PROGRAM F15_CaseControlCACData
VAR
	rtrigScanBarcode			: R_TRIG;
	fbScannerCtrl				: FB_SCANNER_CameraSelect;
	bScanCaseLabel				: BOOL;
	fbCaseLableEvaluation		: FB_SCANNER_Evaluation;

	rtrigSetCaseValidationOK	: R_TRIG;
	rtrigSetCaseValidationNOK	: R_TRIG;

	sCaseSerialCode				: T_CASE_Barcode;
	sFirstOuterInCase			: T_OUTER_Barcode;
	sLastOuterInCase			: T_OUTER_Barcode;
	sFirstPackSerialCode		: T_PACK_Barcode;
	sLastPackSerialCode			: T_PACK_Barcode;


	fbSequenceControl			: FB_SYSTEM_SeqControl;
	nSequenceStep				: INT;
	b00_Idle					: BOOL;
	b01_ScanLabel				: BOOL;
	b03_CreateFileName			: BOOL;
	b05_MoveCaseData			: BOOL;
	b08_WriteFSSFile			: BOOL;
	b10_CaseTraceValid			: BOOL;
	b18_CaseValid				: BOOL;
	b19_CaseInvalid				: BOOL;
	b20_Done					: BOOL;

	bDone						: BOOL;
	bBusy						: BOOL;
	tonScanTimeout				: TON;
	tonOverTime					: TON;

	rtrigCACData				: R_TRIG;
	tF15TimeExecution			: TIME;
	bTestSeq					: BOOL;
	sCACFileTemplate			: T_CAC_Filename;

	stValidateCACData			: ST_CAC_Data;
	fbMoveCaseData				: FB_CASE_ValidatePrintCACData;

	sPrintCaseContent			: STRING(255);

	fbPopulateCHMData				: FB_CHM_PopulateDataForFSS3;
	fbWriteCHMFile				: FB_CHM_WriteFSS3Files; (*Old system supporting FSS2 -> FB_CHM_WriteFSSFile;*)

	fbWriteCACToArchiveDB			: FB_CAC_WriteHierachyToDB;
	fbCaseStatusPulse				: TON;
	bCACValid					: BOOL;
	bCHMValid					: BOOL;


	fbMoveVerifiedCAC				: FB_CASE_MoveVerifiedCAC;
	fbMoveFailedCAC				: FB_CASE_MoveFailedCAC;

	fbCaseEfficiency				: FB_KPI_GenericEfficiency;
	fbCaseInspectionEfficiency		: FB_KPI_CaseEfficiency;
	(*fbCaseInspectionEfficiency		: FB_KPI_PACAN_CaseEfficiency;*)
	fbRejectCount					: CTU;
	nRejectActualCount				: WORD;

	fbCaseValidationScanned			: FB_CTU32;
	fbCaseValidationCorrect			: FB_CTU32;
	fbCaseValidationNoCaseLabel		: FB_CTU32;
	fbCaseValidationCasePackerReject	: FB_CTU32;

	aLastCaseBarcodes				: ARRAY[1..cMAX_LAST_CASE_BARCODES] OF T_CASE_Barcode;
	fbAddVerifiedCaseBarcode		: FB_CASE_AddVerifiedCaseBarcode;

	fbCaseLevelCounter	: FB_KPI_CaseLevelCounter;
	tofCaseValidationCameraOFFDelay 	: TOF;

	fbFileWriteCACError				: FB_LOG_FileWriteError;
	fbFileWriteCHMError			: FB_LOG_FileWriteError;

END_VAR
(*
VAR CONSTANT
	sOptions						: ST_SCANNER_Options := (eScannerType := E_MV_440SR_FULL, nImageBuffer := 1, nExpectedResp := 1);
END_VAR*)
VAR // added by the converter: edge detectors and wires of the graphical bodies
    _w1, _w2, _w3, _w4 : BOOL;
END_VAR

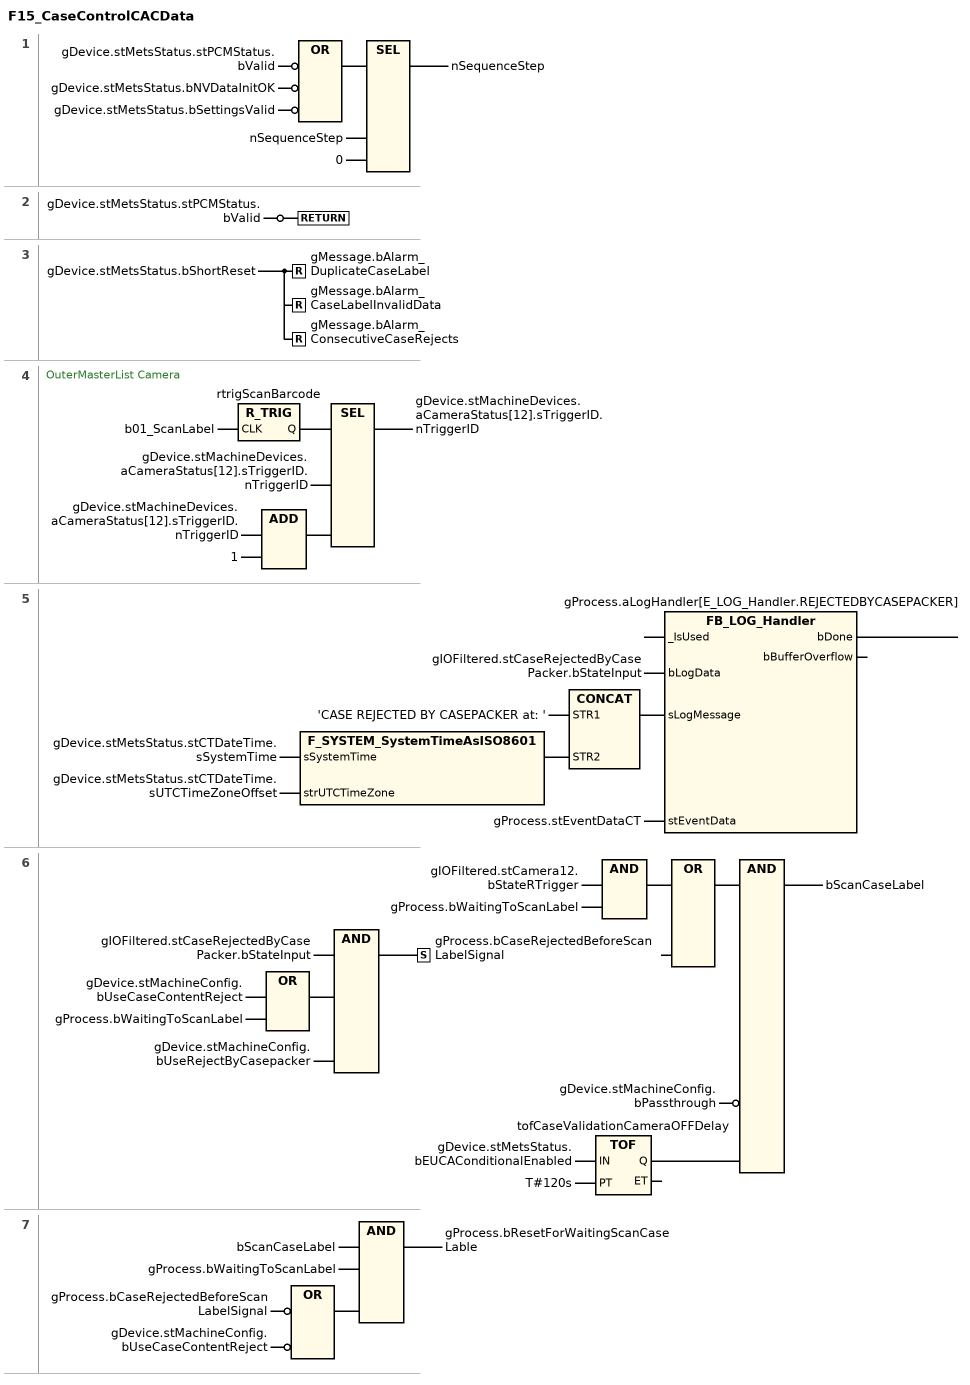
// NETWORK 1
nSequenceStep := SEL(NOT gDevice.stMetsStatus.stPCMStatus.bValid OR NOT gDevice.stMetsStatus.bNVDataInitOK OR NOT gDevice.stMetsStatus.bSettingsValid, nSequenceStep, 0);

// NETWORK 2
IF NOT gDevice.stMetsStatus.stPCMStatus.bValid THEN RETURN; END_IF

// NETWORK 3
gMessage.bAlarm_DuplicateCaseLabel R= gDevice.stMetsStatus.bShortReset;
gMessage.bAlarm_CaseLabelInvalidData R= gDevice.stMetsStatus.bShortReset;
gMessage.bAlarm_ConsecutiveCaseRejects R= gDevice.stMetsStatus.bShortReset;

// NETWORK 4
// OuterMasterList Camera
rtrigScanBarcode(CLK := b01_ScanLabel); // R_TRIG
gDevice.stMachineDevices.aCameraStatus[12].sTriggerID.nTriggerID := SEL(rtrigScanBarcode.Q, gDevice.stMachineDevices.aCameraStatus[12].sTriggerID.nTriggerID, gDevice.stMachineDevices.aCameraStatus[12].sTriggerID.nTriggerID + 1);

// NETWORK 5
gProcess.aLogHandler[E_LOG_Handler.REJECTEDBYCASEPACKER](
    bLogData := gIOFiltered.stCaseRejectedByCasePacker.bStateInput,
    sLogMessage := CONCAT(STR1 := 'CASE REJECTED BY CASEPACKER at: ', STR2 := F_SYSTEM_SystemTimeAsISO8601(sSystemTime := gDevice.stMetsStatus.stCTDateTime.sSystemTime, strUTCTimeZone := gDevice.stMetsStatus.stCTDateTime.sUTCTimeZoneOffset)),
    stEventData := gProcess.stEventDataCT); // FB_LOG_Handler

// NETWORK 6
_w2 := gIOFiltered.stCamera12.bStateRTrigger AND gProcess.bWaitingToScanLabel;
_w1 := gIOFiltered.stCaseRejectedByCasePacker.bStateInput AND (gDevice.stMachineConfig.bUseCaseContentReject OR gProcess.bWaitingToScanLabel) AND gDevice.stMachineConfig.bUseRejectByCasepacker;
gProcess.bCaseRejectedBeforeScanLabelSignal S= _w1;
tofCaseValidationCameraOFFDelay(IN := gDevice.stMetsStatus.bEUCAConditionalEnabled, PT := T#120s); // TOF
bScanCaseLabel := (_w2 OR _w1) AND NOT gDevice.stMachineConfig.bPassthrough AND tofCaseValidationCameraOFFDelay.Q;

// NETWORK 7
gProcess.bResetForWaitingScanCaseLable := bScanCaseLabel AND gProcess.bWaitingToScanLabel AND (NOT gProcess.bCaseRejectedBeforeScanLabelSignal OR NOT gDevice.stMachineConfig.bUseCaseContentReject);

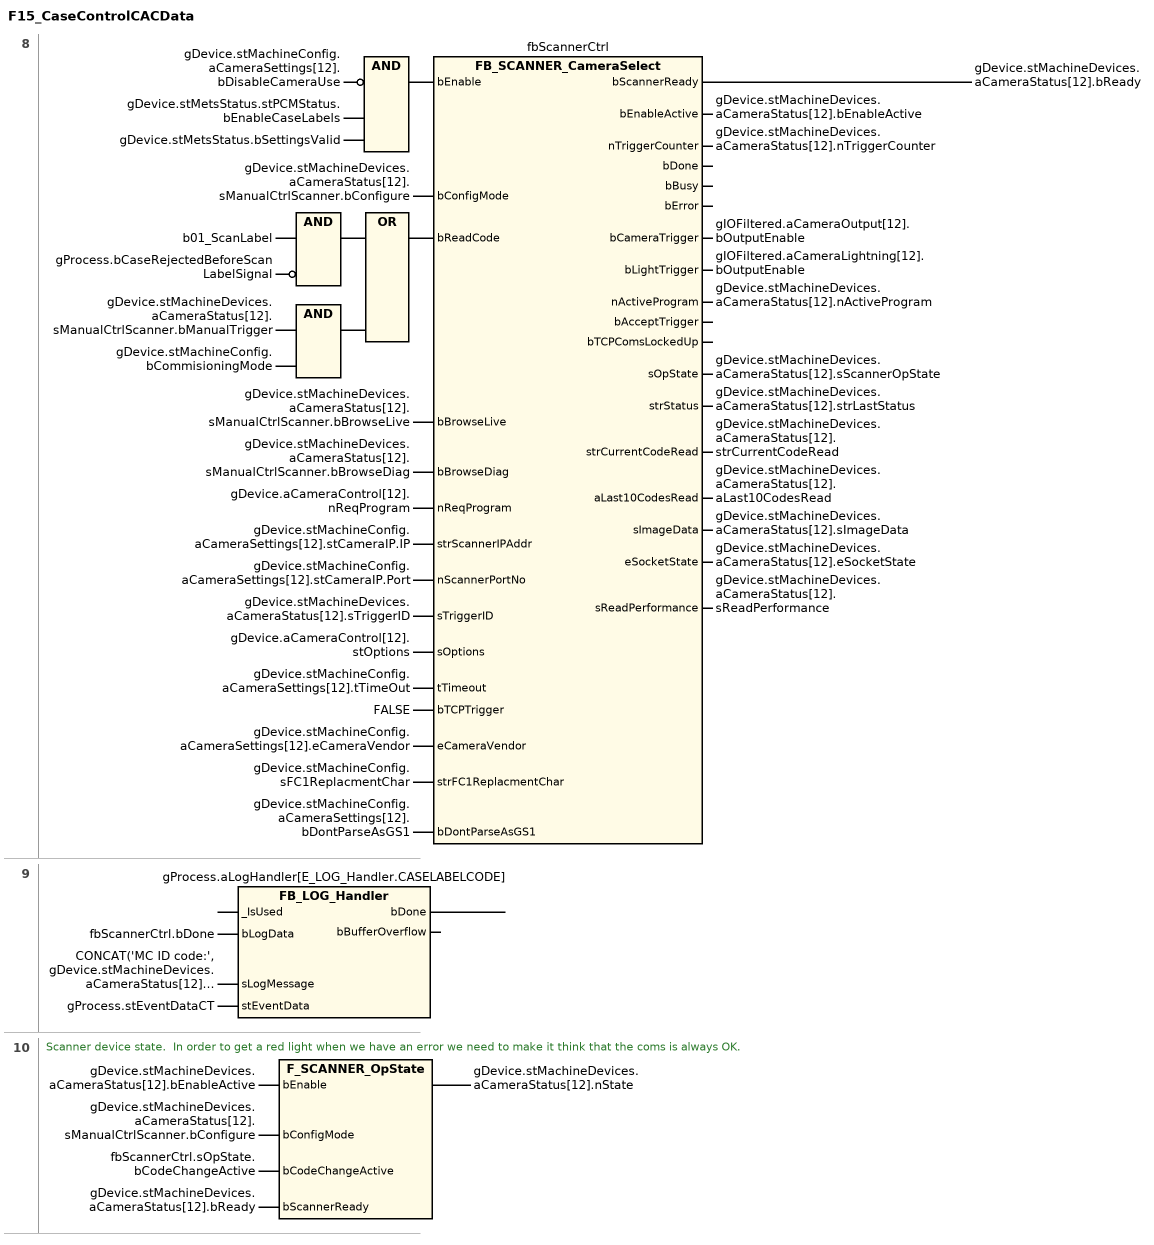
// NETWORK 8
fbScannerCtrl(
    bEnable := NOT gDevice.stMachineConfig.aCameraSettings[12].bDisableCameraUse AND gDevice.stMetsStatus.stPCMStatus.bEnableCaseLabels AND gDevice.stMetsStatus.bSettingsValid,
    bConfigMode := gDevice.stMachineDevices.aCameraStatus[12].sManualCtrlScanner.bConfigure,
    bReadCode := b01_ScanLabel AND NOT gProcess.bCaseRejectedBeforeScanLabelSignal OR gDevice.stMachineDevices.aCameraStatus[12].sManualCtrlScanner.bManualTrigger AND gDevice.stMachineConfig.bCommisioningMode,
    bBrowseLive := gDevice.stMachineDevices.aCameraStatus[12].sManualCtrlScanner.bBrowseLive,
    bBrowseDiag := gDevice.stMachineDevices.aCameraStatus[12].sManualCtrlScanner.bBrowseDiag,
    nReqProgram := gDevice.aCameraControl[12].nReqProgram,
    strScannerIPAddr := gDevice.stMachineConfig.aCameraSettings[12].stCameraIP.IP,
    nScannerPortNo := gDevice.stMachineConfig.aCameraSettings[12].stCameraIP.Port,
    sTriggerID := gDevice.stMachineDevices.aCameraStatus[12].sTriggerID,
    sOptions := gDevice.aCameraControl[12].stOptions,
    tTimeout := gDevice.stMachineConfig.aCameraSettings[12].tTimeOut,
    bTCPTrigger := FALSE,
    eCameraVendor := gDevice.stMachineConfig.aCameraSettings[12].eCameraVendor,
    strFC1ReplacmentChar := gDevice.stMachineConfig.sFC1ReplacmentChar,
    bDontParseAsGS1 := gDevice.stMachineConfig.aCameraSettings[12].bDontParseAsGS1,
    bEnableActive => gDevice.stMachineDevices.aCameraStatus[12].bEnableActive,
    nTriggerCounter => gDevice.stMachineDevices.aCameraStatus[12].nTriggerCounter,
    bCameraTrigger => gIOFiltered.aCameraOutput[12].bOutputEnable,
    bLightTrigger => gIOFiltered.aCameraLightning[12].bOutputEnable,
    nActiveProgram => gDevice.stMachineDevices.aCameraStatus[12].nActiveProgram,
    sOpState => gDevice.stMachineDevices.aCameraStatus[12].sScannerOpState,
    strStatus => gDevice.stMachineDevices.aCameraStatus[12].strLastStatus,
    strCurrentCodeRead => gDevice.stMachineDevices.aCameraStatus[12].strCurrentCodeRead,
    aLast10CodesRead => gDevice.stMachineDevices.aCameraStatus[12].aLast10CodesRead,
    sImageData => gDevice.stMachineDevices.aCameraStatus[12].sImageData,
    eSocketState => gDevice.stMachineDevices.aCameraStatus[12].eSocketState,
    sReadPerformance => gDevice.stMachineDevices.aCameraStatus[12].sReadPerformance); // FB_SCANNER_CameraSelect
gDevice.stMachineDevices.aCameraStatus[12].bReady := fbScannerCtrl.bScannerReady;

// NETWORK 9
gProcess.aLogHandler[E_LOG_Handler.CASELABELCODE](
    bLogData := fbScannerCtrl.bDone,
    sLogMessage := CONCAT('MC ID code:', gDevice.stMachineDevices.aCameraStatus[12].strCurrentCodeRead),
    stEventData := gProcess.stEventDataCT); // FB_LOG_Handler

// NETWORK 10
// Scanner device state.  In order to get a red light when we have an error we need to make it think that the coms is always OK.
gDevice.stMachineDevices.aCameraStatus[12].nState := F_SCANNER_OpState(bEnable := gDevice.stMachineDevices.aCameraStatus[12].bEnableActive, bConfigMode := gDevice.stMachineDevices.aCameraStatus[12].sManualCtrlScanner.bConfigure, bCodeChangeActive := fbScannerCtrl.sOpState.bCodeChangeActive, bScannerReady := gDevice.stMachineDevices.aCameraStatus[12].bReady);

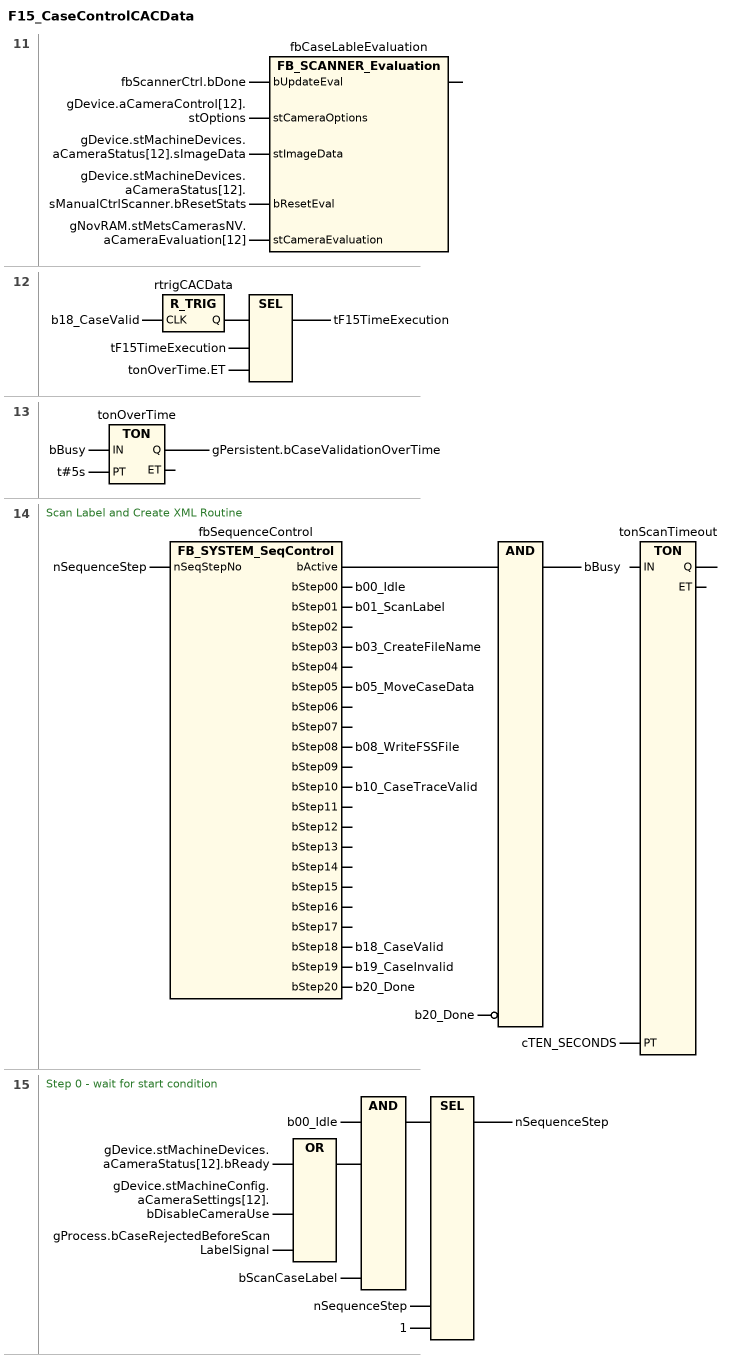
// NETWORK 11
fbCaseLableEvaluation(
    bUpdateEval := fbScannerCtrl.bDone,
    stCameraOptions := gDevice.aCameraControl[12].stOptions,
    stImageData := gDevice.stMachineDevices.aCameraStatus[12].sImageData,
    bResetEval := gDevice.stMachineDevices.aCameraStatus[12].sManualCtrlScanner.bResetStats,
    stCameraEvaluation := gNovRAM.stMetsCamerasNV.aCameraEvaluation[12]); // FB_SCANNER_Evaluation

// NETWORK 12
rtrigCACData(CLK := b18_CaseValid); // R_TRIG
tF15TimeExecution := SEL(rtrigCACData.Q, tF15TimeExecution, tonOverTime.ET);

// NETWORK 13
tonOverTime(IN := bBusy, PT := t#5s); // TON
gPersistent.bCaseValidationOverTime := tonOverTime.Q;

// NETWORK 14
// 					Scan Label and Create XML Routine
//
//
//
fbSequenceControl(
    nSeqStepNo := nSequenceStep,
    bStep00 => b00_Idle,
    bStep01 => b01_ScanLabel,
    bStep03 => b03_CreateFileName,
    bStep05 => b05_MoveCaseData,
    bStep08 => b08_WriteFSSFile,
    bStep10 => b10_CaseTraceValid,
    bStep18 => b18_CaseValid,
    bStep19 => b19_CaseInvalid,
    bStep20 => b20_Done); // FB_SYSTEM_SeqControl
_w3 := fbSequenceControl.bActive AND NOT b20_Done;
bBusy := _w3;
tonScanTimeout(IN := _w3, PT := cTEN_SECONDS); // TON

// NETWORK 15
// 					Step 0 - wait for start condition
//
//
nSequenceStep := SEL(b00_Idle AND (gDevice.stMachineDevices.aCameraStatus[12].bReady OR gDevice.stMachineConfig.aCameraSettings[12].bDisableCameraUse OR gProcess.bCaseRejectedBeforeScanLabelSignal) AND bScanCaseLabel, nSequenceStep, 1);

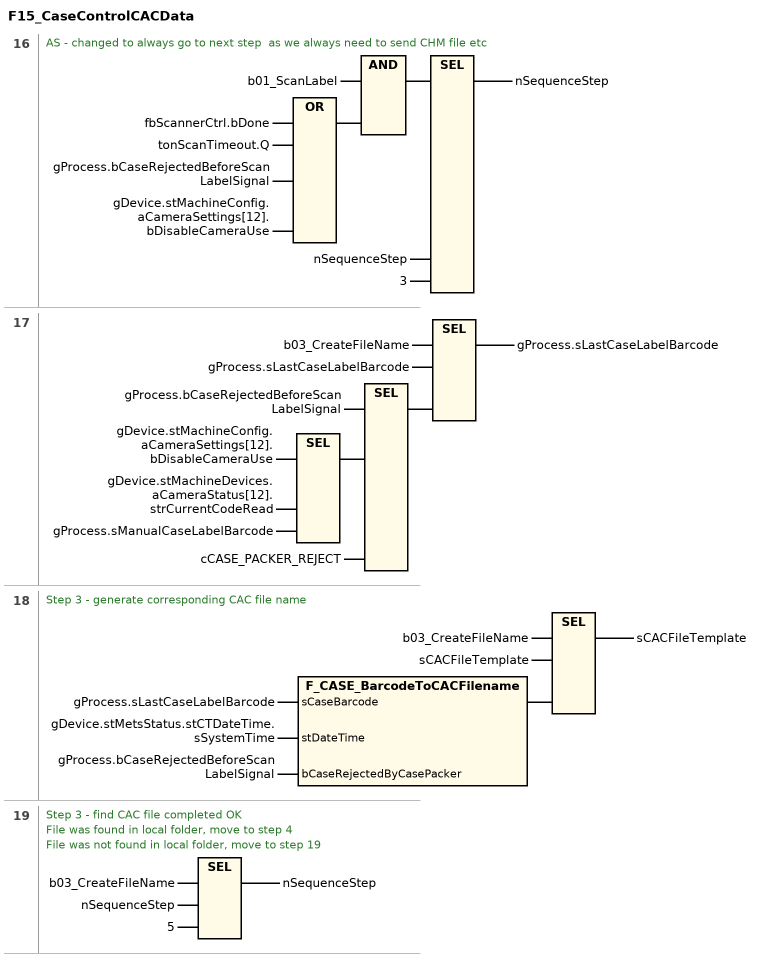
// NETWORK 16
// 					AS - changed to always go to next step  as we always need to send CHM file etc
//
//
nSequenceStep := SEL(b01_ScanLabel AND (fbScannerCtrl.bDone OR tonScanTimeout.Q OR gProcess.bCaseRejectedBeforeScanLabelSignal OR gDevice.stMachineConfig.aCameraSettings[12].bDisableCameraUse), nSequenceStep, 3);

// NETWORK 17
gProcess.sLastCaseLabelBarcode := SEL(b03_CreateFileName, gProcess.sLastCaseLabelBarcode, SEL(gProcess.bCaseRejectedBeforeScanLabelSignal, SEL(gDevice.stMachineConfig.aCameraSettings[12].bDisableCameraUse, gDevice.stMachineDevices.aCameraStatus[12].strCurrentCodeRead, gProcess.sManualCaseLabelBarcode), cCASE_PACKER_REJECT));

// NETWORK 18
// Step 3 - generate corresponding CAC file name
sCACFileTemplate := SEL(b03_CreateFileName, sCACFileTemplate, F_CASE_BarcodeToCACFilename(sCaseBarcode := gProcess.sLastCaseLabelBarcode, stDateTime := gDevice.stMetsStatus.stCTDateTime.sSystemTime, bCaseRejectedByCasePacker := gProcess.bCaseRejectedBeforeScanLabelSignal));

// NETWORK 19
// 					Step 3 - find CAC file completed OK
// File was found in local folder, move to step 4
// File was not found in local folder, move to step 19
//
nSequenceStep := SEL(b03_CreateFileName, nSequenceStep, 5);

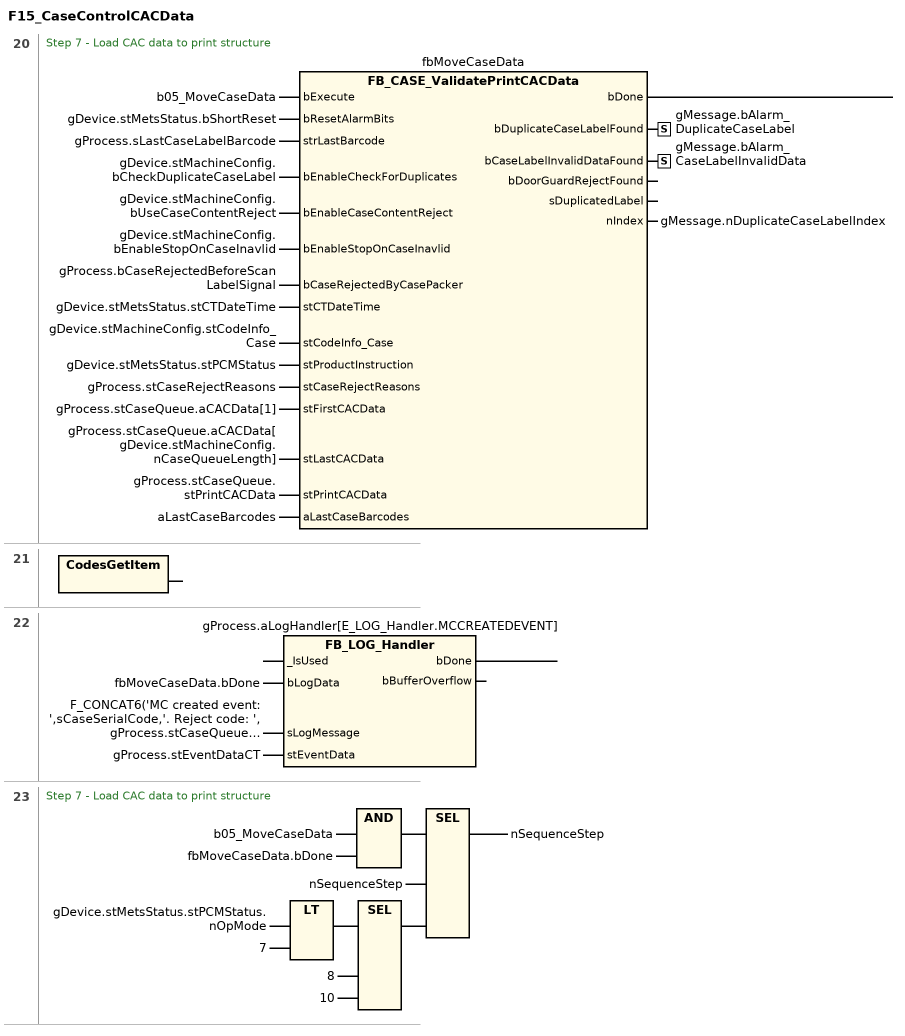
// NETWORK 20
// Step 7 - Load CAC data to print structure
fbMoveCaseData(
    bExecute := b05_MoveCaseData,
    bResetAlarmBits := gDevice.stMetsStatus.bShortReset,
    strLastBarcode := gProcess.sLastCaseLabelBarcode,
    bEnableCheckForDuplicates := gDevice.stMachineConfig.bCheckDuplicateCaseLabel,
    bEnableCaseContentReject := gDevice.stMachineConfig.bUseCaseContentReject,
    bEnableStopOnCaseInavlid := gDevice.stMachineConfig.bEnableStopOnCaseInavlid,
    bCaseRejectedByCasePacker := gProcess.bCaseRejectedBeforeScanLabelSignal,
    stCTDateTime := gDevice.stMetsStatus.stCTDateTime,
    stCodeInfo_Case := gDevice.stMachineConfig.stCodeInfo_Case,
    stProductInstruction := gDevice.stMetsStatus.stPCMStatus,
    stCaseRejectReasons := gProcess.stCaseRejectReasons,
    stFirstCACData := gProcess.stCaseQueue.aCACData[1],
    stLastCACData := gProcess.stCaseQueue.aCACData[gDevice.stMachineConfig.nCaseQueueLength],
    stPrintCACData := gProcess.stCaseQueue.stPrintCACData,
    aLastCaseBarcodes := aLastCaseBarcodes,
    nIndex => gMessage.nDuplicateCaseLabelIndex); // FB_CASE_ValidatePrintCACData
gMessage.bAlarm_DuplicateCaseLabel S= fbMoveCaseData.bDuplicateCaseLabelFound;
gMessage.bAlarm_CaseLabelInvalidData S= fbMoveCaseData.bCaseLabelInvalidDataFound;

// NETWORK 21
CodesGetItem();

// NETWORK 22
gProcess.aLogHandler[E_LOG_Handler.MCCREATEDEVENT](
    bLogData := fbMoveCaseData.bDone,
    sLogMessage := F_CONCAT6('MC created event: ',sCaseSerialCode,'. Reject code: ', gProcess.stCaseQueue.stPrintCACData.CaseRejectCode,', with case content: ', sPrintCaseContent),
    stEventData := gProcess.stEventDataCT); // FB_LOG_Handler

// NETWORK 23
// 					Step 7 - Load CAC data to print structure
//
//
nSequenceStep := SEL(b05_MoveCaseData AND fbMoveCaseData.bDone, nSequenceStep, SEL(gDevice.stMetsStatus.stPCMStatus.nOpMode < 7, 8, 10));

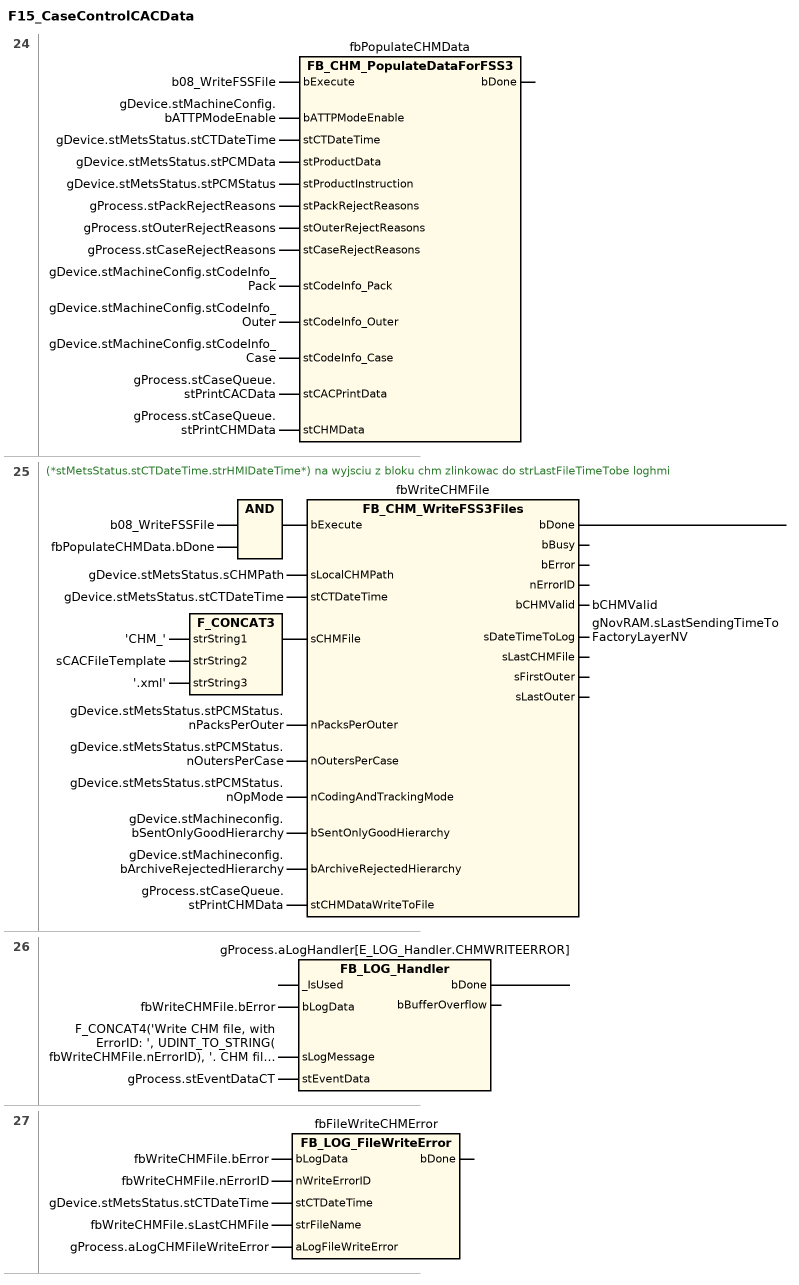
// NETWORK 24
fbPopulateCHMData(
    bExecute := b08_WriteFSSFile,
    bATTPModeEnable := gDevice.stMachineConfig.bATTPModeEnable,
    stCTDateTime := gDevice.stMetsStatus.stCTDateTime,
    stProductData := gDevice.stMetsStatus.stPCMData,
    stProductInstruction := gDevice.stMetsStatus.stPCMStatus,
    stPackRejectReasons := gProcess.stPackRejectReasons,
    stOuterRejectReasons := gProcess.stOuterRejectReasons,
    stCaseRejectReasons := gProcess.stCaseRejectReasons,
    stCodeInfo_Pack := gDevice.stMachineConfig.stCodeInfo_Pack,
    stCodeInfo_Outer := gDevice.stMachineConfig.stCodeInfo_Outer,
    stCodeInfo_Case := gDevice.stMachineConfig.stCodeInfo_Case,
    stCACPrintData := gProcess.stCaseQueue.stPrintCACData,
    stCHMData := gProcess.stCaseQueue.stPrintCHMData); // FB_CHM_PopulateDataForFSS3

// NETWORK 25
// (*stMetsStatus.stCTDateTime.strHMIDateTime*) na wyjsciu z bloku chm zlinkowac do strLastFileTimeTobe loghmi
fbWriteCHMFile(
    bExecute := b08_WriteFSSFile AND fbPopulateCHMData.bDone,
    sLocalCHMPath := gDevice.stMetsStatus.sCHMPath,
    stCTDateTime := gDevice.stMetsStatus.stCTDateTime,
    sCHMFile := F_CONCAT3(strString1 := 'CHM_', strString2 := sCACFileTemplate, strString3 := '.xml'),
    nPacksPerOuter := gDevice.stMetsStatus.stPCMStatus.nPacksPerOuter,
    nOutersPerCase := gDevice.stMetsStatus.stPCMStatus.nOutersPerCase,
    nCodingAndTrackingMode := gDevice.stMetsStatus.stPCMStatus.nOpMode,
    bSentOnlyGoodHierarchy := gDevice.stMachineconfig.bSentOnlyGoodHierarchy,
    bArchiveRejectedHierarchy := gDevice.stMachineconfig.bArchiveRejectedHierarchy,
    stCHMDataWriteToFile := gProcess.stCaseQueue.stPrintCHMData,
    bCHMValid => bCHMValid,
    sDateTimeToLog => gNovRAM.sLastSendingTimeToFactoryLayerNV); // FB_CHM_WriteFSS3Files

// NETWORK 26
gProcess.aLogHandler[E_LOG_Handler.CHMWRITEERROR](
    bLogData := fbWriteCHMFile.bError,
    sLogMessage := F_CONCAT4('Write CHM file, with ErrorID: ', UDINT_TO_STRING(fbWriteCHMFile.nErrorID), '. CHM file name: ', fbWriteCHMFile.sCHMFile),
    stEventData := gProcess.stEventDataCT); // FB_LOG_Handler

// NETWORK 27
fbFileWriteCHMError(
    bLogData := fbWriteCHMFile.bError,
    nWriteErrorID := fbWriteCHMFile.nErrorID,
    stCTDateTime := gDevice.stMetsStatus.stCTDateTime,
    strFileName := fbWriteCHMFile.sLastCHMFile,
    aLogFileWriteError := gProcess.aLogCHMFileWriteError); // FB_LOG_FileWriteError

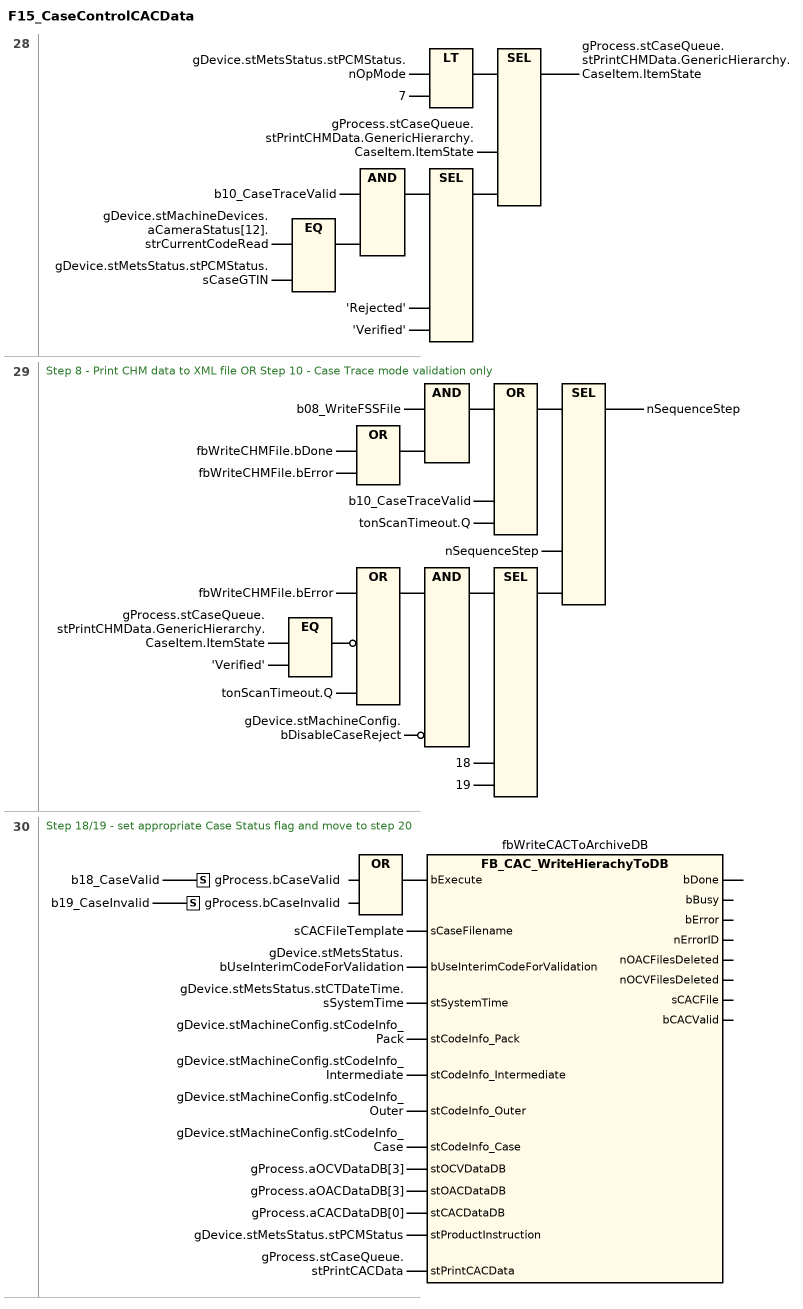
// NETWORK 28
gProcess.stCaseQueue.stPrintCHMData.GenericHierarchy.CaseItem.ItemState := SEL(gDevice.stMetsStatus.stPCMStatus.nOpMode < 7, gProcess.stCaseQueue.stPrintCHMData.GenericHierarchy.CaseItem.ItemState, SEL(b10_CaseTraceValid AND gDevice.stMachineDevices.aCameraStatus[12].strCurrentCodeRead = gDevice.stMetsStatus.stPCMStatus.sCaseGTIN, 'Rejected', 'Verified'));

// NETWORK 29
// Step 8 - Print CHM data to XML file OR Step 10 - Case Trace mode validation only
nSequenceStep := SEL(b08_WriteFSSFile AND (fbWriteCHMFile.bDone OR fbWriteCHMFile.bError) OR b10_CaseTraceValid OR tonScanTimeout.Q, nSequenceStep, SEL((fbWriteCHMFile.bError OR NOT (gProcess.stCaseQueue.stPrintCHMData.GenericHierarchy.CaseItem.ItemState = 'Verified') OR tonScanTimeout.Q) AND NOT gDevice.stMachineConfig.bDisableCaseReject, 18, 19));

// NETWORK 30
// Step 18/19 - set appropriate Case Status flag and move to step 20
gProcess.bCaseValid S= b18_CaseValid;
gProcess.bCaseInvalid S= b19_CaseInvalid;
fbWriteCACToArchiveDB(
    bExecute := b18_CaseValid OR b19_CaseInvalid,
    sCaseFilename := sCACFileTemplate,
    bUseInterimCodeForValidation := gDevice.stMetsStatus.bUseInterimCodeForValidation,
    stSystemTime := gDevice.stMetsStatus.stCTDateTime.sSystemTime,
    stCodeInfo_Pack := gDevice.stMachineConfig.stCodeInfo_Pack,
    stCodeInfo_Intermediate := gDevice.stMachineConfig.stCodeInfo_Intermediate,
    stCodeInfo_Outer := gDevice.stMachineConfig.stCodeInfo_Outer,
    stCodeInfo_Case := gDevice.stMachineConfig.stCodeInfo_Case,
    stOCVDataDB := gProcess.aOCVDataDB[3],
    stOACDataDB := gProcess.aOACDataDB[3],
    stCACDataDB := gProcess.aCACDataDB[0],
    stProductInstruction := gDevice.stMetsStatus.stPCMStatus,
    stPrintCACData := gProcess.stCaseQueue.stPrintCACData); // FB_CAC_WriteHierachyToDB

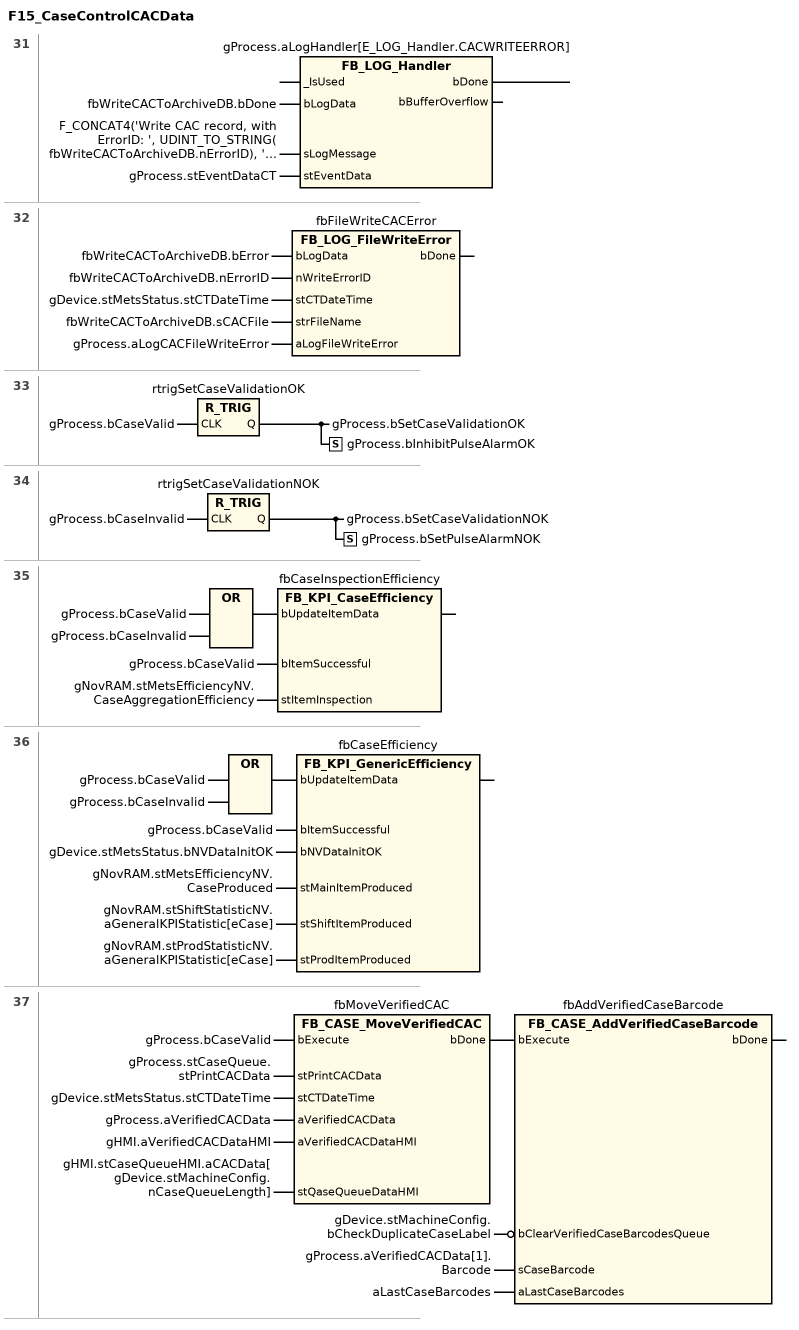
// NETWORK 31
gProcess.aLogHandler[E_LOG_Handler.CACWRITEERROR](
    bLogData := fbWriteCACToArchiveDB.bDone,
    sLogMessage := F_CONCAT4('Write CAC record, with ErrorID: ', UDINT_TO_STRING(fbWriteCACToArchiveDB.nErrorID), '. CAC file name: ', fbWriteCACToArchiveDB.sCACFile),
    stEventData := gProcess.stEventDataCT); // FB_LOG_Handler

// NETWORK 32
fbFileWriteCACError(
    bLogData := fbWriteCACToArchiveDB.bError,
    nWriteErrorID := fbWriteCACToArchiveDB.nErrorID,
    stCTDateTime := gDevice.stMetsStatus.stCTDateTime,
    strFileName := fbWriteCACToArchiveDB.sCACFile,
    aLogFileWriteError := gProcess.aLogCACFileWriteError); // FB_LOG_FileWriteError

// NETWORK 33
rtrigSetCaseValidationOK(CLK := gProcess.bCaseValid); // R_TRIG
gProcess.bSetCaseValidationOK := rtrigSetCaseValidationOK.Q;
gProcess.bInhibitPulseAlarmOK S= rtrigSetCaseValidationOK.Q;

// NETWORK 34
rtrigSetCaseValidationNOK(CLK := gProcess.bCaseInvalid); // R_TRIG
gProcess.bSetCaseValidationNOK := rtrigSetCaseValidationNOK.Q;
gProcess.bSetPulseAlarmNOK S= rtrigSetCaseValidationNOK.Q;

// NETWORK 35
fbCaseInspectionEfficiency(
    bUpdateItemData := gProcess.bCaseValid OR gProcess.bCaseInvalid,
    bItemSuccessful := gProcess.bCaseValid,
    stItemInspection := gNovRAM.stMetsEfficiencyNV.CaseAggregationEfficiency); // FB_KPI_CaseEfficiency

// NETWORK 36
fbCaseEfficiency(
    bUpdateItemData := gProcess.bCaseValid OR gProcess.bCaseInvalid,
    bItemSuccessful := gProcess.bCaseValid,
    bNVDataInitOK := gDevice.stMetsStatus.bNVDataInitOK,
    stMainItemProduced := gNovRAM.stMetsEfficiencyNV.CaseProduced,
    stShiftItemProduced := gNovRAM.stShiftStatisticNV.aGeneralKPIStatistic[eCase],
    stProdItemProduced := gNovRAM.stProdStatisticNV.aGeneralKPIStatistic[eCase]); // FB_KPI_GenericEfficiency

// NETWORK 37
fbMoveVerifiedCAC(
    bExecute := gProcess.bCaseValid,
    stPrintCACData := gProcess.stCaseQueue.stPrintCACData,
    stCTDateTime := gDevice.stMetsStatus.stCTDateTime,
    aVerifiedCACData := gProcess.aVerifiedCACData,
    aVerifiedCACDataHMI := gHMI.aVerifiedCACDataHMI,
    stQaseQueueDataHMI := gHMI.stCaseQueueHMI.aCACData[gDevice.stMachineConfig.nCaseQueueLength]); // FB_CASE_MoveVerifiedCAC
fbAddVerifiedCaseBarcode(
    bExecute := fbMoveVerifiedCAC.bDone,
    bClearVerifiedCaseBarcodesQueue := NOT gDevice.stMachineConfig.bCheckDuplicateCaseLabel,
    sCaseBarcode := gProcess.aVerifiedCACData[1].Barcode,
    aLastCaseBarcodes := aLastCaseBarcodes); // FB_CASE_AddVerifiedCaseBarcode

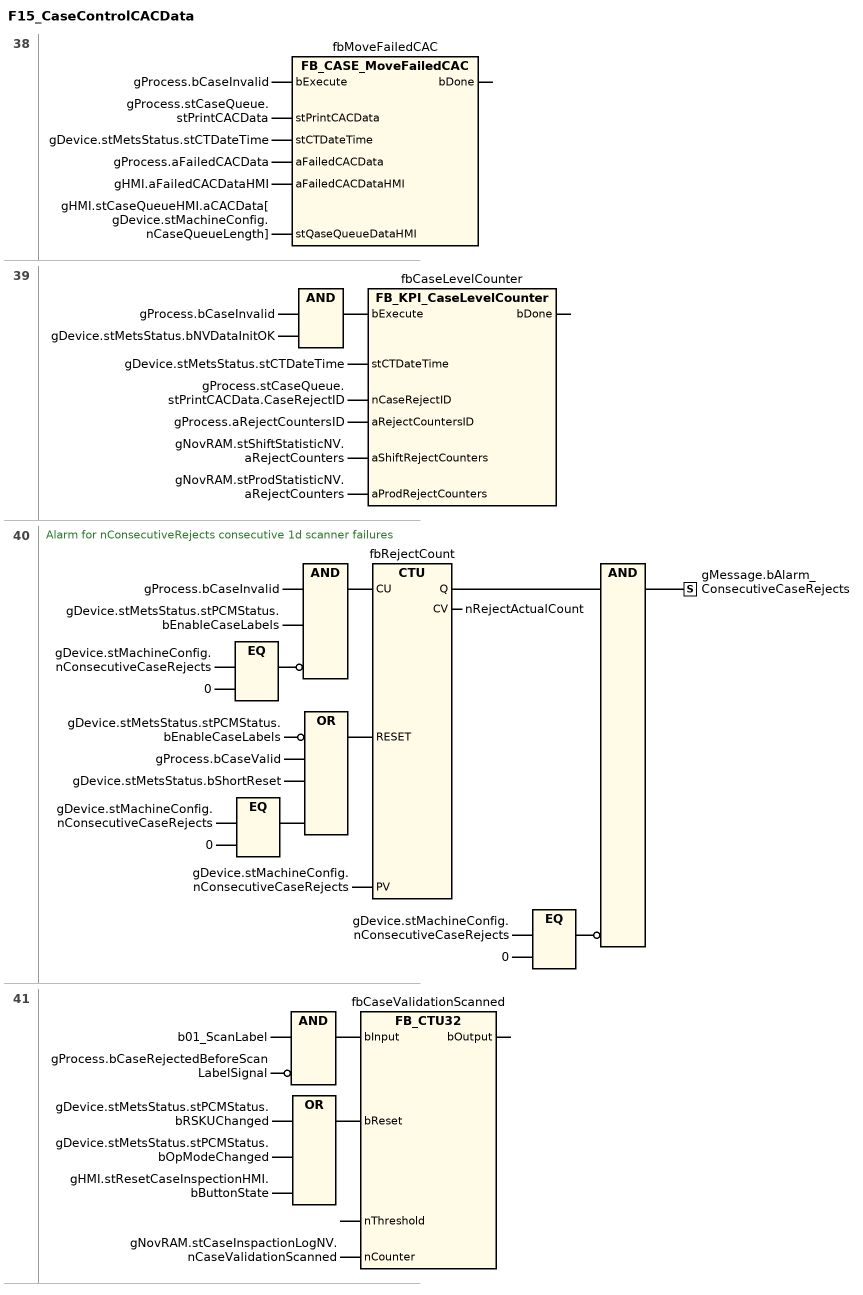
// NETWORK 38
fbMoveFailedCAC(
    bExecute := gProcess.bCaseInvalid,
    stPrintCACData := gProcess.stCaseQueue.stPrintCACData,
    stCTDateTime := gDevice.stMetsStatus.stCTDateTime,
    aFailedCACData := gProcess.aFailedCACData,
    aFailedCACDataHMI := gHMI.aFailedCACDataHMI,
    stQaseQueueDataHMI := gHMI.stCaseQueueHMI.aCACData[gDevice.stMachineConfig.nCaseQueueLength]); // FB_CASE_MoveFailedCAC

// NETWORK 39
fbCaseLevelCounter(
    bExecute := gProcess.bCaseInvalid AND gDevice.stMetsStatus.bNVDataInitOK,
    stCTDateTime := gDevice.stMetsStatus.stCTDateTime,
    nCaseRejectID := gProcess.stCaseQueue.stPrintCACData.CaseRejectID,
    aRejectCountersID := gProcess.aRejectCountersID,
    aShiftRejectCounters := gNovRAM.stShiftStatisticNV.aRejectCounters,
    aProdRejectCounters := gNovRAM.stProdStatisticNV.aRejectCounters); // FB_KPI_CaseLevelCounter

// NETWORK 40
// Alarm for nConsecutiveRejects consecutive 1d scanner failures
fbRejectCount(
    CU := gProcess.bCaseInvalid AND gDevice.stMetsStatus.stPCMStatus.bEnableCaseLabels AND NOT (gDevice.stMachineConfig.nConsecutiveCaseRejects = 0),
    RESET := NOT gDevice.stMetsStatus.stPCMStatus.bEnableCaseLabels OR gProcess.bCaseValid OR gDevice.stMetsStatus.bShortReset OR gDevice.stMachineConfig.nConsecutiveCaseRejects = 0,
    PV := gDevice.stMachineConfig.nConsecutiveCaseRejects,
    CV => nRejectActualCount); // CTU
gMessage.bAlarm_ConsecutiveCaseRejects S= fbRejectCount.Q AND NOT (gDevice.stMachineConfig.nConsecutiveCaseRejects = 0);

// NETWORK 41
fbCaseValidationScanned(
    bInput := b01_ScanLabel AND NOT gProcess.bCaseRejectedBeforeScanLabelSignal,
    bReset := gDevice.stMetsStatus.stPCMStatus.bRSKUChanged OR gDevice.stMetsStatus.stPCMStatus.bOpModeChanged OR gHMI.stResetCaseInspectionHMI.bButtonState,
    nCounter := gNovRAM.stCaseInspactionLogNV.nCaseValidationScanned); // FB_CTU32

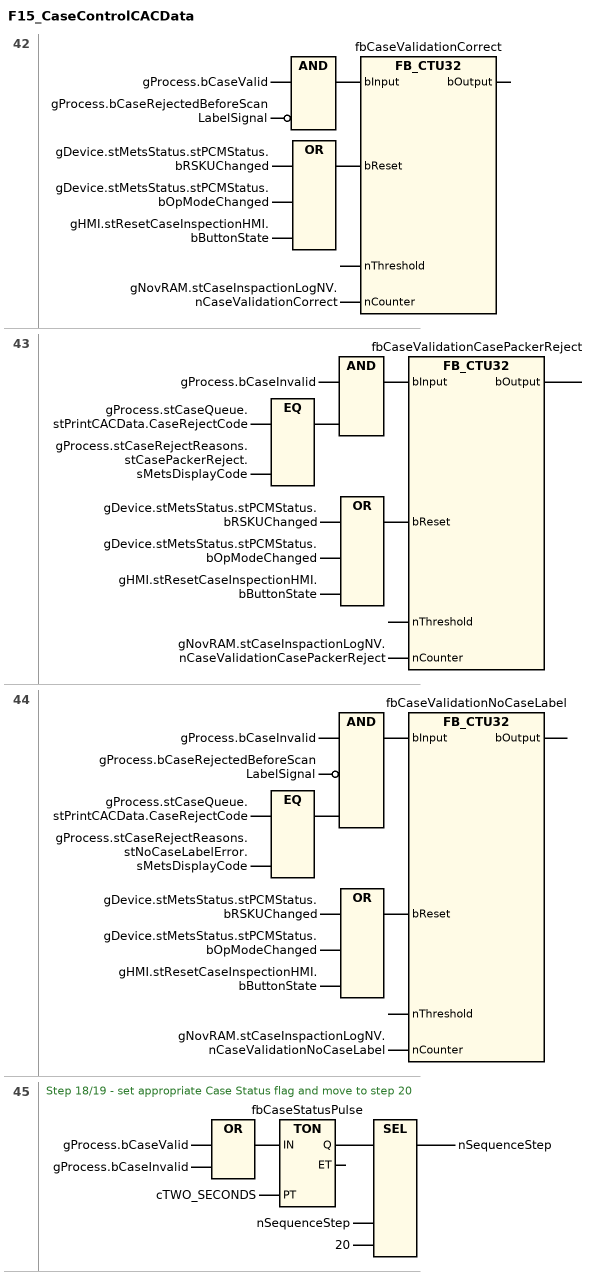
// NETWORK 42
fbCaseValidationCorrect(
    bInput := gProcess.bCaseValid AND NOT gProcess.bCaseRejectedBeforeScanLabelSignal,
    bReset := gDevice.stMetsStatus.stPCMStatus.bRSKUChanged OR gDevice.stMetsStatus.stPCMStatus.bOpModeChanged OR gHMI.stResetCaseInspectionHMI.bButtonState,
    nCounter := gNovRAM.stCaseInspactionLogNV.nCaseValidationCorrect); // FB_CTU32

// NETWORK 43
fbCaseValidationCasePackerReject(
    bInput := gProcess.bCaseInvalid AND gProcess.stCaseQueue.stPrintCACData.CaseRejectCode = gProcess.stCaseRejectReasons.stCasePackerReject.sMetsDisplayCode,
    bReset := gDevice.stMetsStatus.stPCMStatus.bRSKUChanged OR gDevice.stMetsStatus.stPCMStatus.bOpModeChanged OR gHMI.stResetCaseInspectionHMI.bButtonState,
    nCounter := gNovRAM.stCaseInspactionLogNV.nCaseValidationCasePackerReject); // FB_CTU32

// NETWORK 44
fbCaseValidationNoCaseLabel(
    bInput := gProcess.bCaseInvalid AND NOT gProcess.bCaseRejectedBeforeScanLabelSignal AND gProcess.stCaseQueue.stPrintCACData.CaseRejectCode = gProcess.stCaseRejectReasons.stNoCaseLabelError.sMetsDisplayCode,
    bReset := gDevice.stMetsStatus.stPCMStatus.bRSKUChanged OR gDevice.stMetsStatus.stPCMStatus.bOpModeChanged OR gHMI.stResetCaseInspectionHMI.bButtonState,
    nCounter := gNovRAM.stCaseInspactionLogNV.nCaseValidationNoCaseLabel); // FB_CTU32

// NETWORK 45
// Step 18/19 - set appropriate Case Status flag and move to step 20
fbCaseStatusPulse(IN := gProcess.bCaseValid OR gProcess.bCaseInvalid, PT := cTWO_SECONDS); // TON
nSequenceStep := SEL(fbCaseStatusPulse.Q, nSequenceStep, 20);

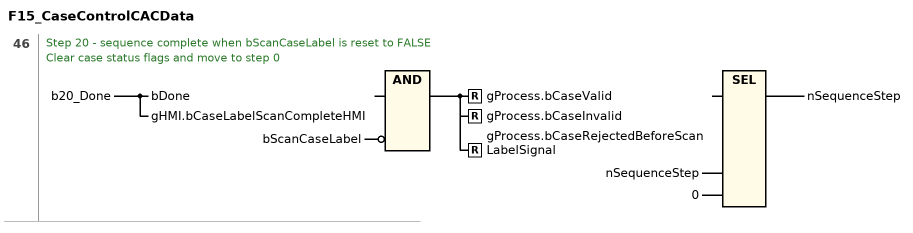
// NETWORK 46
// 					Step 20 - sequence complete when bScanCaseLabel is reset to FALSE
// Clear case status flags and move to step 0
//
bDone := b20_Done;
gHMI.bCaseLabelScanCompleteHMI := b20_Done;
_w4 := b20_Done AND NOT bScanCaseLabel;
gProcess.bCaseValid R= _w4;
gProcess.bCaseInvalid R= _w4;
gProcess.bCaseRejectedBeforeScanLabelSignal R= _w4;
nSequenceStep := SEL(_w4, nSequenceStep, 0);

ACTION CodesGetItem:
IF gDevice.stMetsStatus.stPCMStatus.nOutersPerCase > 0 AND gDevice.stMetsStatus.stPCMStatus.nPacksPerOuter > 0 THEN

	sCaseSerialCode := F_CODE_GetItem(gProcess.stCaseQueue.stPrintCACData.Barcode, eCodeAIType.SerialCode, gDevice.stMachineConfig.stCodeInfo_Case);
	sFirstOuterInCase := F_CODE_GetItem(gProcess.stCaseQueue.stPrintCACData.Outer[1].Barcode, eCodeAIType.SerialCode, gDevice.stMachineConfig.stCodeInfo_Outer);
	sLastOuterInCase := F_CODE_GetItem(gProcess.stCaseQueue.stPrintCACData.Outer[gDevice.stMetsStatus.stPCMStatus.nOutersPerCase].Barcode, eCodeAIType.SerialCode, gDevice.stMachineConfig.stCodeInfo_Outer);
	sFirstPackSerialCode := F_CODE_GetItem(gProcess.stCaseQueue.stPrintCACData.Outer[1].PackCode[1], eCodeAIType.SerialCode, gDevice.stMachineConfig.stCodeInfo_Pack);
	sLastPackSerialCode := F_CODE_GetItem(gProcess.stCaseQueue.stPrintCACData.Outer[gDevice.stMetsStatus.stPCMStatus.nOutersPerCase].PackCode[gDevice.stMetsStatus.stPCMStatus.nPacksPerOuter], eCodeAIType.SerialCode, gDevice.stMachineConfig.stCodeInfo_Pack);

	sFirstOuterInCase	:= RIGHT(sFirstOuterInCase,7);
	sLastOuterInCase	:= RIGHT(sLastOuterInCase,7);
	sFirstPackSerialCode	:= RIGHT(sFirstPackSerialCode,7);
	sLastPackSerialCode	:= RIGHT(sLastPackSerialCode,7);

	sPrintCaseContent  := F_CONCAT9('Init OUT ID [',sFirstOuterInCase, '] ; Last OUT ID [', sLastOuterInCase,  '] ; Init PK ID [',sFirstPackSerialCode, '] ; Last PK ID [', sLastPackSerialCode,']');
END_IF
END_ACTION

END_PROGRAM

(* stored: Version 1.1.0.1
   POU F15_CaseControlCACData: Id {6995a318-9841-4988-a699-2b329bc50f2b}, SpecialFunc None
   Action CodesGetItem: Id {b7ba0711-cdec-4b42-82f6-a2fe6a70881d} *)
